TYPE DUT_HMI EXTENDS DUT_Control_Base :
STRUCT
	ModeValue : INT:= 1; // 0: Manual; 1: Auto;
	DisableAutoManual : BOOL;
END_STRUCT
END_TYPE

(* stored: Version 1.1.0.1, ProductVersion 3.1.4024.12
   DUT DUT_HMI: Id {bc4f9921-1dd7-45e9-9775-32ca85304546} *)
